Staubli VAL3: ModbusGet.pgx

program modbusGet(num& x_nResult (dimensions=1))
begin
  if (dStartControl[1]==true and dStartControl[2]==false and dStartControl[3]==false)
    x_nResult=1
  elseIf (dStartControl[1]==false and dStartControl[2]==true and dStartControl[3]==false)
    x_nResult=2
  elseIf (dStartControl[1]==false and dStartControl[2]==false and dStartControl[3]==true)
    x_nResult=3
  else
    x_nResult=0
  endIf
end
